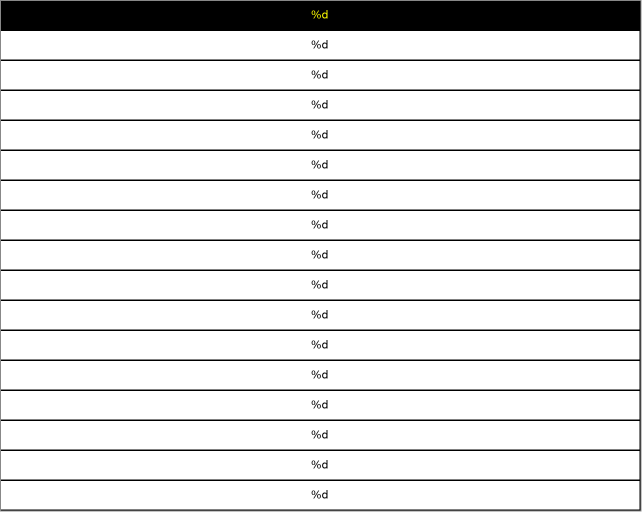
VISUALIZATION CARTON_FILLING_SHIFT_ELEMENT  // 642x512
VAR_INPUT
	index:		UDINT;
END_VAR
    Rectangle (0,0 640x30), "%d", text variable: wu_cartonForming_shiftRegister_debug.shift_debug[index].step_id
    Rectangle (0,30 640x30), "%d", text variable: wu_cartonFilling_shiftRegister_debug.shift_debug[index].status.0, colour toggle: wu_cartonFilling_shiftRegister_debug.shift_debug[index].status.0
    Rectangle (0,90 640x30), "%d", text variable: wu_cartonFilling_shiftRegister_debug.shift_debug[index].reject_reason
    Rectangle (0,120 640x30), "%d", text variable: wu_cartonFilling_shiftRegister_debug.shift_debug[index].status.4, colour toggle: wu_cartonFilling_shiftRegister_debug.shift_debug[index].status.4
    Rectangle (0,180 640x30), "%d", text variable: wu_cartonFilling_shiftRegister_debug.shift_debug[index].status.11, colour toggle: wu_cartonFilling_shiftRegister_debug.shift_debug[index].status.11
    Rectangle (0,150 640x30), "%d", text variable: wu_cartonFilling_shiftRegister_debug.shift_debug[index].status.10, colour toggle: wu_cartonFilling_shiftRegister_debug.shift_debug[index].status.10
    Rectangle (0,60 640x30), "%d", text variable: wu_cartonFilling_shiftRegister_debug.shift_debug[index].status.1, colour toggle: wu_cartonFilling_shiftRegister_debug.shift_debug[index].status.1
    Rectangle (0,210 640x30), "%d", text variable: wu_cartonFilling_shiftRegister_debug.shift_debug[index].status.12, colour toggle: wu_cartonFilling_shiftRegister_debug.shift_debug[index].status.12
    Rectangle (0,240 640x30), "%d", text variable: wu_cartonFilling_shiftRegister_debug.shift_debug[index].status.13, colour toggle: wu_cartonFilling_shiftRegister_debug.shift_debug[index].status.13
    Rectangle (0,270 640x30), "%d", text variable: wu_cartonFilling_shiftRegister_debug.shift_debug[index].status.14, colour toggle: wu_cartonFilling_shiftRegister_debug.shift_debug[index].status.14
    Rectangle (0,300 640x30), "%d", text variable: wu_cartonFilling_shiftRegister_debug.shift_debug[index].status.15, colour toggle: wu_cartonFilling_shiftRegister_debug.shift_debug[index].status.15
    Rectangle (0,330 640x30), "%d", text variable: wu_cartonFilling_shiftRegister_debug.shift_debug[index]._1st_layer_robot_id
    Rectangle (0,360 640x30), "%d", text variable: wu_cartonFilling_shiftRegister_debug.shift_debug[index]._2nd_layer_robot_id
    Rectangle (0,390 640x30), "%d", text variable: wu_cartonFilling_shiftRegister_debug.shift_debug[index]._3rd_layer_robot_id
    Rectangle (0,420 640x30), "%d", text variable: wu_cartonFilling_shiftRegister_debug.shift_debug[index]._4th_layer_robot_id
    Rectangle (0,450 640x30), "%d", text variable: wu_cartonFilling_shiftRegister_debug.shift_debug[index]._5th_layer_robot_id
    Rectangle (0,480 640x30), "%d", text variable: wu_cartonFilling_shiftRegister_debug.shift_debug[index]._6th_layer_robot_id
END_VISUALIZATION

(* stored: Version 1.1.0.1, ProductVersion 3.1.4024.3
   Visu CARTON_FILLING_SHIFT_ELEMENT: Id {72f29a0c-4196-4b29-b2ae-90b1c85f8d92} *)
